INTERFACE I_RpcDynamicConfigAmsNetId

METHOD WithAmsNetId : I_RpcDynamicConfigAmsPort
VAR_INPUT
	sAmsNetId	: T_AmsNetID;
END_VAR
END_METHOD

END_INTERFACE

(* stored: Version 1.1.0.1, ProductVersion 3.1.4024.12
   Itf I_RpcDynamicConfigAmsNetId: Id {adfddc74-34fd-459e-bf15-06f40b585475}
   Method WithAmsNetId: Id {035089dd-f095-4a6e-8c35-e63df558f6bb} *)
